// TIA Portal project "rilevamento_colori" (V16)

(* hardware
DEVICE "S71500/ET200MP station_1"  S7-1500 station
   slot 0: "Telaio di montaggio_0"  Rack  6ES7 590-1***0-0AA0
   slot 1: "PLC_1"  CPU 1512C-1 PN  6ES7 512-1CK01-0AB0  V2.8
      slot 3: "Display CPU_1"  6ES7591-1AA00-0AA0
      slot 32768: "Interfaccia PROFINET_1"  X1
         slot 32769: "Porta_1"  X1 P1
         slot 32770: "Porta_2"  X1 P2
      slot 34817: "Virtual CP interface port_1"  Virtual CP interface port  Virtual CP interface port
*)

// ===== PLC "PLC_1"  CPU 1512C-1 PN =====

VAR_GLOBAL   // PLC tag table "Tabella delle variabili standard"
   "red" AT %MW0 : Int;   // variabile contenente la quantità di rosso (red)
   "green" AT %MW10 : Int;   // variabile contenente la quantità di verde (green)
   "blue" AT %MW20 : Int;   // variabile contenente la quantità di blu (blue)
END_VAR

DATA_BLOCK "DB_Prova"   // DB1
{ S7_Optimized_Access := 'TRUE' }
VERSION : 0.1
   VAR
      colore : String;   // variabile contenente il colore (stringa)
   END_VAR
BEGIN
END_DATA_BLOCK

ORGANIZATION_BLOCK "Main"   // OB1, LAD, ProgramCycle
TITLE = "Main Program Sweep (Cycle)"
{ S7_Optimized_Access := 'TRUE' }
VERSION : 0.1
   VAR_INPUT
      Initial_Call : Bool;   // Initial call of this OB
      Remanence : Bool;   // =True, if remanent data are available
   END_VAR
BEGIN
END_ORGANIZATION_BLOCK